// TIA Portal V20 export
TYPE "LER_TypeFATModeInterface"
// stored: Access Published
   STRUCT
      HoursTest : "LER_TypeFATMode_HoursTest";
      Capability : "LER_TypeFATMode_Capability";
      Sampling : "LER_TypeFATMode_Sampling";
   END_STRUCT;
END_TYPE
